// TIA Portal V19 export
VAR_GLOBAL   // PLC tag table "14_Settings"
END_VAR
VAR_GLOBAL CONSTANT   // user constants
   MAX_NO_OF_DEVICES : Int := 10;
   MAX_NO_OF_MODULES : Int := 10;
END_VAR
